// TIA Portal V16 export
// export: Created 2021-04-09T13:38:05.7500687Z, ExportSetting WithDefaults, DisplayName Totally Integrated Automation Portal, DisplayVersion V16, DisplayName TIA Portal Version Control Interface, DisplayVersion V16, DisplayName TIA Portal Openness, DisplayVersion V16, DisplayName STEP 7 Professional, DisplayVersion V16, DisplayName STEP 7 Safety, DisplayVersion V16, DisplayName WinCC Unified SCADA Engineering System, DisplayVersion V16
FUNCTION "alarmBlock" : Void   // FC10, LAD
{ S7_Optimized_Access := 'TRUE' }
VERSION : 0.1
// stored: AutoNumber true, IsIECCheckEnabled false, SetENOAutomatically false, UDAEnableTagReadback false
   VAR_TEMP
      i : DInt;
   END_VAR
BEGIN

REGION Network 1: Тепловое реле Конв1
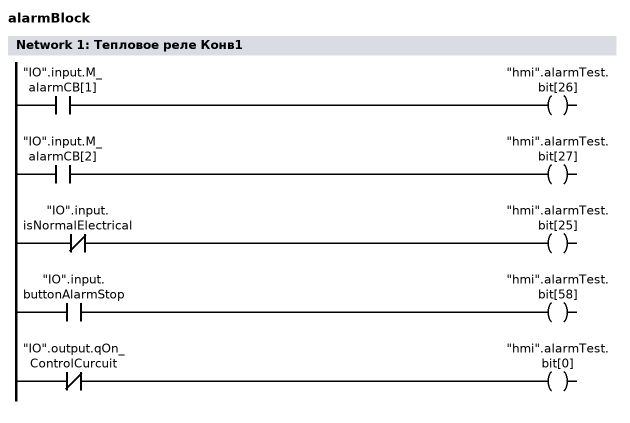
   RUNG wire#powerrail
      Contact( "IO".input.M_alarmCB[1] )
      Coil( "hmi".alarmTest.bit[26] )
   END_RUNG
   RUNG wire#powerrail
      Contact( "IO".input.M_alarmCB[2] )
      Coil( "hmi".alarmTest.bit[27] )
   END_RUNG
   RUNG wire#powerrail
      I_Contact( "IO".input.isNormalElectrical )
      Coil( "hmi".alarmTest.bit[25] )
   END_RUNG
   RUNG wire#powerrail
      Contact( "IO".input.buttonAlarmStop )
      Coil( "hmi".alarmTest.bit[58] )
   END_RUNG
   RUNG wire#powerrail
      I_Contact( "IO".output.qOn_ControlCurcuit )
      Coil( "hmi".alarmTest.bit[0] )
   END_RUNG
   // the same network as SCL:
   "hmi".alarmTest.bit[26] := "IO".input.M_alarmCB[1];
   "hmi".alarmTest.bit[27] := "IO".input.M_alarmCB[2];
   "hmi".alarmTest.bit[25] := NOT "IO".input.isNormalElectrical;
   "hmi".alarmTest.bit[58] := "IO".input.buttonAlarmStop;
   "hmi".alarmTest.bit[0] := NOT "IO".output.qOn_ControlCurcuit;
END_REGION

REGION Network 2 (SCL): обрывы весовых датчиков
   #i := 0;
   FOR #i := 1 TO 12 DO
       IF "signalKVSStation".currentWeight[#i] > 7000 THEN
           "hmi".alarmTest.bit[12 + #i] := true;
       ELSE
           "hmi".alarmTest.bit[12 + #i] := false;
       END_IF;
   END_FOR;
END_REGION

REGION Network 3 (SCL)
   #i := 0;
   FOR #i := 0 TO 70 DO
       IF "hmi".alarmTest.bit[#i] THEN
           "hmi".commonAlarm := true;
           EXIT;
       END_IF;
       IF #i = 70 THEN
           "hmi".commonAlarm := false;
       END_IF;
   END_FOR;
END_REGION
END_FUNCTION
